{attribute 'GeneratedUsingTerminal: ELM9410-0000-0016'}
{attribute addProperty BoxType "ELM9410-0000-0016"}
{attribute addProperty Id "StatusAT %I*Status_06143A9F4"}
{attribute addProperty CRC "2104461108"}
{attribute addProperty Size "4"}
TYPE MMS_Device_Inputs_7D6F8734 :
STRUCT
	{attribute addProperty Name "Status"}
	Status AT %I* : Status_06143A9F;
END_STRUCT
END_TYPE

(* stored: Version 1.2.0.0, ProductVersion 3.1.4024.9
   DUT MMS_Device_Inputs_7D6F8734: Id {f71d32d0-fcd6-42d1-9e62-f4ec1b5d2804} *)
